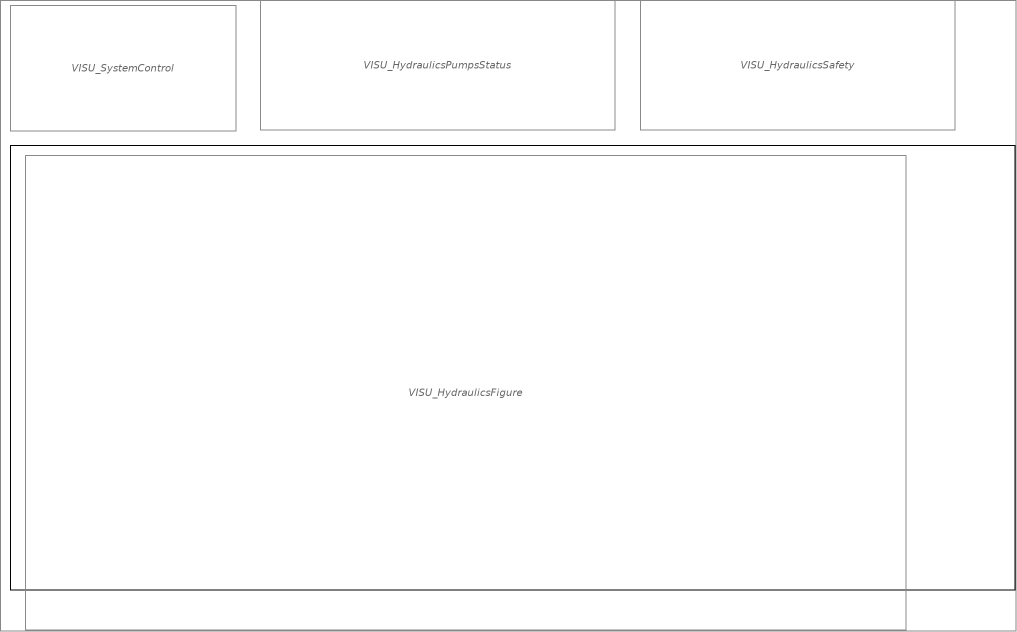
VISUALIZATION VISU_HydraulicsOverview  // 1017x632
VAR_IN_OUT
	ref : Hydraulics;
    widget : HydraulicsWidget;
    ref_safety : SafetyHydraulics;
END_VAR
    Rectangle (10,145 1005x445)
    Frame (10,5 226x126)
        shows VISU_SystemControl(status := widget.actualStatus, button_initialize := widget.button_initialize, button_operating := widget.button_operating, button_locking := widget.button_locking)
    Frame (25,155 881x475)
        shows VISU_HydraulicsFigure(ref := ref, widget := widget, ref_safety := ref_safety)
    Frame (260,0 355x130)
        shows VISU_HydraulicsPumpsStatus(ref := ref, widget := widget, ref_safety := ref_safety)
    Frame (640,0 315x130)
        shows VISU_HydraulicsSafety(ref := ref, widget := widget, ref_safety := ref_safety)
END_VISUALIZATION

(* stored: Version 1.1.0.1, ProductVersion 3.1.4019.2
   Visu VISU_HydraulicsOverview: Id {34da9c2f-7af3-4705-8466-188f055a5b53} *)
